PROGRAM MAIN
VAR
	myStructTypeVar : StructType;
	counter : DINT;
END_VAR

myStructTypeVar.enumTypeVariable := EnumType.member2;
counter := counter + 1;

END_PROGRAM

(* stored: Version 1.1.0.1, ProductVersion 3.1.4024.15
   POU MAIN: Id {313d875a-09d8-412f-8daa-90367b1d5c09}, SpecialFunc None *)
